// TIA Portal V21 export
VAR_GLOBAL   // PLC tag table "K_TipoLetturaScrittura"
END_VAR
VAR_GLOBAL CONSTANT   // user constants
   K_TipoLetturaScrittura_SolaLettura : Int := 0;
   K_TipoLetturaScrittura_SolaScrittura : Int := 1;
   K_TipoLetturaScrittura_LetturaScrittura : Int := 2;
   K_TipoLetturaScrittura_NessunaLetturaScrittura : Int := 3;
END_VAR
